{attribute 'GeneratedUsingTerminal: EL3423-0000-0016'}
{attribute addProperty BoxType "EL3423-0000-0016"}
{attribute addProperty Id "PQF_AvgAT %I*REAL4PQF_MinAT %I*REAL4PQF_MaxAT %I*REAL4"}
{attribute addProperty CRC "3760468548"}
{attribute addProperty Size "12"}
TYPE Total_Statistic_PQF_E0243244 EXTENDS InputBase_8311D824 :
STRUCT
	{attribute addProperty Name "PQF_Avg"}
	PQF_Avg AT %I* : REAL;
	{attribute addProperty Name "PQF_Min"}
	PQF_Min AT %I* : REAL;
	{attribute addProperty Name "PQF_Max"}
	PQF_Max AT %I* : REAL;
END_STRUCT
END_TYPE

(* stored: Version 1.2.0.0, ProductVersion 3.1.4024.9
   DUT Total_Statistic_PQF_E0243244: Id {1cef8cd7-c86e-4fbb-a966-76b974ddf2ad} *)
